KUKA KRL program: traccionv1.src, traccionv1.dat

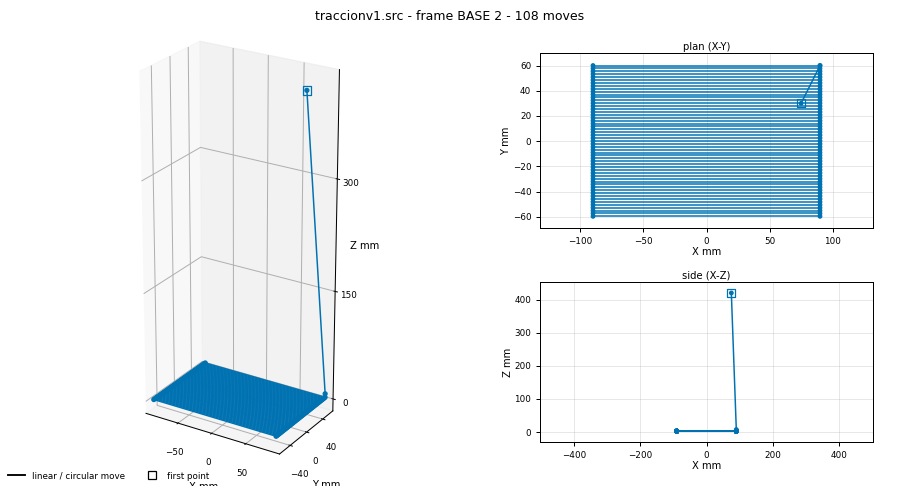
[picture p0: tool path of traccionv1.src in frame BASE 2, 108 of 110 moves have a stored position in this frame; points joined in program order, loops and branches not executed]
--- traccionv1.src ---
&ACCESS RVP
&PARAM TEMPLATE = C:\KRC\Roboter\Template\vorgabe
&PARAM EDITMASK = *
DEF traccionv1( )
;FOLD INI;%{PE}%V3.2.0,%MKUKATPBASIS,%CINIT,%VCOMMON,%P
;FOLD BAS INI;%{E}%V3.2.0,%MKUKATPBASIS,%CINIT,%VINIT,%P
GLOBAL INTERRUPT DECL 3 WHEN $STOPMESS==TRUE DO IR_STOPM ( )
INTERRUPT ON 3
BAS (#INITMOV,0 )
;ENDFOLD (BAS INI)
;FOLD A20 INI;%{E}%V3.2.0,%MKUKATPA20,%CINIT,%VINIT,%P
IF ARC20==TRUE THEN
A20 (ARC_INI)
INTERRUPT DECL 6 WHEN $CYCFLAG[3]==FALSE DO A20(TECH_STOP2)
ENDIF
;ENDFOLD (A20 INI)
;FOLD A10 INI;%{E}%V3.2.0,%MKUKATPARC,%CINIT,%VINIT,%P
IF A10_OPTION==#ACTIVE THEN
INTERRUPT DECL 4 WHEN $CYCFLAG[2]==FALSE DO A10 (#APPL_ERROR)
INTERRUPT DECL 7 WHEN A_ARC_SWI==#ACTIVE DO A10 (#ARC_SEAM)
INTERRUPT DECL 5 WHEN A_FLY_ARC==TRUE DO A10 (#HPU_ARC)
INTERRUPT  ON 5
A10_INI ( )
ENDIF
;ENDFOLD (A10 INI)
;FOLD GRIPPER INI;%{E}%V3.2.0,%MKUKATPGRIPPER,%CINIT,%VINIT,%P
USER_GRP(0,DUMMY,DUMMY,GDEFAULT)
;ENDFOLD (GRIPPER INI)
;FOLD SPOT INI;%{E}%V3.2.0,%MKUKATPSPOT,%CINIT,%VINIT,%P
USERSPOT(#INIT)
;ENDFOLD (SPOT INI)
;FOLD TOUCHSENSE INI;%{E}%V3.2.0,%MKUKATPTS,%CINIT,%VINIT,%P
IF H70_OPTION THEN
INTERRUPT DECL 15 WHEN $MEAS_PULSE[TOUCH_I[TOUCH_ACTIVE].IN_NR] DO H70 (6,CD0 )
INTERRUPT DECL 16 WHEN $ZERO_MOVE DO H70 (7,CD0 )
INTERRUPT DECL 17 WHEN $TECHPAR_C[FG_TOUCH,8]>0.5 DO H70 (8,CD0)
H70 (1,CD0 )
ENDIF
;ENDFOLD (TOUCHSENSE INI)
;FOLD USER INI;%{E}%V3.2.0,%MKUKATPUSER,%CINIT,%VINIT,%P
;Make your modifications here
;ENDFOLD (USER INI)
;ENDFOLD (INI)
; SPEED PTP FOR AXIS
$VEL_AXIS[1] = 15
$VEL_AXIS[2] = 15
$VEL_AXIS[3] = 15
$VEL_AXIS[4] = 15
$VEL_AXIS[5] = 15
$VEL_AXIS[6] = 15
;SMOOTHNESS
$APO.CDIS = 2
;ADVANCE
$ADVANCE = 3
;SET TOOL AND BASE
$TOOL = TOOL_DATA[3]
$BASE = BASE_DATA[2]
;HOME
;FOLD PTP HOME Vel=10% DEFAULT
$BWDSTART=FALSE
$H_POS=XHOME
PDAT_ACT=PDEFAULT
FDAT_ACT=FHOME
BAS(#PTP_DAT )
BAS (#VEL_PTP,10 )
PTP XHOME
;ENDFOLD
;USER PROGRAM
;SPEED $VEL.CP
$VEL.CP=0.045
; OUT[TEMP] = 200
; OUT[vent] = 1
; OUT[RPM] = 45
; USER POSES CALLS
PTP {X 75, Y 30, Z 420, A 0, B 90, C 0}
; USER POSES CALLS
LIN {X 90.0, Y 60.0, Z 7.5, A 0, B 90, C 0} C_DIS
WAIT SEC 1
$OUT[1] = TRUE
LIN {X 90.0, Y 60.0, Z 2.5, A 0, B 90, C 0} C_DIS
LIN {X -90.0, Y 60.0, Z 2.5, A 0, B 90, C 0} C_DIS
LIN {X -90.0, Y 57.7, Z 2.5, A 0, B 90, C 0} C_DIS
LIN {X 90.0, Y 57.7, Z 2.5, A 0, B 90, C 0} C_DIS
LIN {X 90.0, Y 55.4, Z 2.5, A 0, B 90, C 0} C_DIS
LIN {X -90.0, Y 55.4, Z 2.5, A 0, B 90, C 0} C_DIS
LIN {X -90.0, Y 53.1, Z 2.5, A 0, B 90, C 0} C_DIS
LIN {X 90.0, Y 53.1, Z 2.5, A 0, B 90, C 0} C_DIS
LIN {X 90.0, Y 50.8, Z 2.5, A 0, B 90, C 0} C_DIS
LIN {X -90.0, Y 50.8, Z 2.5, A 0, B 90, C 0} C_DIS
LIN {X -90.0, Y 48.5, Z 2.5, A 0, B 90, C 0} C_DIS
LIN {X 90.0, Y 48.5, Z 2.5, A 0, B 90, C 0} C_DIS
LIN {X 90.0, Y 46.2, Z 2.5, A 0, B 90, C 0} C_DIS
LIN {X -90.0, Y 46.2, Z 2.5, A 0, B 90, C 0} C_DIS
LIN {X -90.0, Y 43.9, Z 2.5, A 0, B 90, C 0} C_DIS
LIN {X 90.0, Y 43.9, Z 2.5, A 0, B 90, C 0} C_DIS
LIN {X 90.0, Y 41.6, Z 2.5, A 0, B 90, C 0} C_DIS
LIN {X -90.0, Y 41.6, Z 2.5, A 0, B 90, C 0} C_DIS
LIN {X -90.0, Y 39.3, Z 2.5, A 0, B 90, C 0} C_DIS
LIN {X 90.0, Y 39.3, Z 2.5, A 0, B 90, C 0} C_DIS
LIN {X 90.0, Y 37.0, Z 2.5, A 0, B 90, C 0} C_DIS
LIN {X -90.0, Y 37.0, Z 2.5, A 0, B 90, C 0} C_DIS
LIN {X -90.0, Y 34.7, Z 2.5, A 0, B 90, C 0} C_DIS
LIN {X 90.0, Y 34.7, Z 2.5, A 0, B 90, C 0} C_DIS
LIN {X 90.0, Y 32.4, Z 2.5, A 0, B 90, C 0} C_DIS
LIN {X -90.0, Y 32.4, Z 2.5, A 0, B 90, C 0} C_DIS
LIN {X -90.0, Y 30.1, Z 2.5, A 0, B 90, C 0} C_DIS
LIN {X 90.0, Y 30.1, Z 2.5, A 0, B 90, C 0} C_DIS
LIN {X 90.0, Y 27.8, Z 2.5, A 0, B 90, C 0} C_DIS
LIN {X -90.0, Y 27.8, Z 2.5, A 0, B 90, C 0} C_DIS
LIN {X -90.0, Y 25.5, Z 2.5, A 0, B 90, C 0} C_DIS
LIN {X 90.0, Y 25.5, Z 2.5, A 0, B 90, C 0} C_DIS
LIN {X 90.0, Y 23.2, Z 2.5, A 0, B 90, C 0} C_DIS
LIN {X -90.0, Y 23.2, Z 2.5, A 0, B 90, C 0} C_DIS
LIN {X -90.0, Y 20.9, Z 2.5, A 0, B 90, C 0} C_DIS
LIN {X 90.0, Y 20.9, Z 2.5, A 0, B 90, C 0} C_DIS
LIN {X 90.0, Y 18.6, Z 2.5, A 0, B 90, C 0} C_DIS
LIN {X -90.0, Y 18.6, Z 2.5, A 0, B 90, C 0} C_DIS
LIN {X -90.0, Y 16.3, Z 2.5, A 0, B 90, C 0} C_DIS
LIN {X 90.0, Y 16.3, Z 2.5, A 0, B 90, C 0} C_DIS
LIN {X 90.0, Y 14.0, Z 2.5, A 0, B 90, C 0} C_DIS
LIN {X -90.0, Y 14.0, Z 2.5, A 0, B 90, C 0} C_DIS
LIN {X -90.0, Y 11.7, Z 2.5, A 0, B 90, C 0} C_DIS
LIN {X 90.0, Y 11.7, Z 2.5, A 0, B 90, C 0} C_DIS
LIN {X 90.0, Y 9.4, Z 2.5, A 0, B 90, C 0} C_DIS
LIN {X -90.0, Y 9.4, Z 2.5, A 0, B 90, C 0} C_DIS
LIN {X -90.0, Y 7.1, Z 2.5, A 0, B 90, C 0} C_DIS
LIN {X 90.0, Y 7.1, Z 2.5, A 0, B 90, C 0} C_DIS
LIN {X 90.0, Y 4.8, Z 2.5, A 0, B 90, C 0} C_DIS
LIN {X -90.0, Y 4.8, Z 2.5, A 0, B 90, C 0} C_DIS
LIN {X -90.0, Y 2.5, Z 2.5, A 0, B 90, C 0} C_DIS
LIN {X 90.0, Y 2.5, Z 2.5, A 0, B 90, C 0} C_DIS
LIN {X 90.0, Y 0.2, Z 2.5, A 0, B 90, C 0} C_DIS
LIN {X -90.0, Y 0.2, Z 2.5, A 0, B 90, C 0} C_DIS
LIN {X -90.0, Y -2.1, Z 2.5, A 0, B 90, C 0} C_DIS
LIN {X 90.0, Y -2.1, Z 2.5, A 0, B 90, C 0} C_DIS
LIN {X 90.0, Y -4.4, Z 2.5, A 0, B 90, C 0} C_DIS
LIN {X -90.0, Y -4.4, Z 2.5, A 0, B 90, C 0} C_DIS
LIN {X -90.0, Y -6.7, Z 2.5, A 0, B 90, C 0} C_DIS
LIN {X 90.0, Y -6.7, Z 2.5, A 0, B 90, C 0} C_DIS
LIN {X 90.0, Y -9.0, Z 2.5, A 0, B 90, C 0} C_DIS
LIN {X -90.0, Y -9.0, Z 2.5, A 0, B 90, C 0} C_DIS
LIN {X -90.0, Y -11.3, Z 2.5, A 0, B 90, C 0} C_DIS
LIN {X 90.0, Y -11.3, Z 2.5, A 0, B 90, C 0} C_DIS
LIN {X 90.0, Y -13.6, Z 2.5, A 0, B 90, C 0} C_DIS
LIN {X -90.0, Y -13.6, Z 2.5, A 0, B 90, C 0} C_DIS
LIN {X -90.0, Y -15.9, Z 2.5, A 0, B 90, C 0} C_DIS
LIN {X 90.0, Y -15.9, Z 2.5, A 0, B 90, C 0} C_DIS
LIN {X 90.0, Y -18.2, Z 2.5, A 0, B 90, C 0} C_DIS
LIN {X -90.0, Y -18.2, Z 2.5, A 0, B 90, C 0} C_DIS
LIN {X -90.0, Y -20.5, Z 2.5, A 0, B 90, C 0} C_DIS
LIN {X 90.0, Y -20.5, Z 2.5, A 0, B 90, C 0} C_DIS
LIN {X 90.0, Y -22.8, Z 2.5, A 0, B 90, C 0} C_DIS
LIN {X -90.0, Y -22.8, Z 2.5, A 0, B 90, C 0} C_DIS
LIN {X -90.0, Y -25.1, Z 2.5, A 0, B 90, C 0} C_DIS
LIN {X 90.0, Y -25.1, Z 2.5, A 0, B 90, C 0} C_DIS
LIN {X 90.0, Y -27.4, Z 2.5, A 0, B 90, C 0} C_DIS
LIN {X -90.0, Y -27.4, Z 2.5, A 0, B 90, C 0} C_DIS
LIN {X -90.0, Y -29.7, Z 2.5, A 0, B 90, C 0} C_DIS
LIN {X 90.0, Y -29.7, Z 2.5, A 0, B 90, C 0} C_DIS
LIN {X 90.0, Y -32.0, Z 2.5, A 0, B 90, C 0} C_DIS
LIN {X -90.0, Y -32.0, Z 2.5, A 0, B 90, C 0} C_DIS
LIN {X -90.0, Y -34.3, Z 2.5, A 0, B 90, C 0} C_DIS
LIN {X 90.0, Y -34.3, Z 2.5, A 0, B 90, C 0} C_DIS
LIN {X 90.0, Y -36.6, Z 2.5, A 0, B 90, C 0} C_DIS
LIN {X -90.0, Y -36.6, Z 2.5, A 0, B 90, C 0} C_DIS
LIN {X -90.0, Y -38.9, Z 2.5, A 0, B 90, C 0} C_DIS
LIN {X 90.0, Y -38.9, Z 2.5, A 0, B 90, C 0} C_DIS
LIN {X 90.0, Y -41.2, Z 2.5, A 0, B 90, C 0} C_DIS
LIN {X -90.0, Y -41.2, Z 2.5, A 0, B 90, C 0} C_DIS
LIN {X -90.0, Y -43.5, Z 2.5, A 0, B 90, C 0} C_DIS
LIN {X 90.0, Y -43.5, Z 2.5, A 0, B 90, C 0} C_DIS
LIN {X 90.0, Y -45.8, Z 2.5, A 0, B 90, C 0} C_DIS
LIN {X -90.0, Y -45.8, Z 2.5, A 0, B 90, C 0} C_DIS
LIN {X -90.0, Y -48.1, Z 2.5, A 0, B 90, C 0} C_DIS
LIN {X 90.0, Y -48.1, Z 2.5, A 0, B 90, C 0} C_DIS
LIN {X 90.0, Y -50.4, Z 2.5, A 0, B 90, C 0} C_DIS
LIN {X -90.0, Y -50.4, Z 2.5, A 0, B 90, C 0} C_DIS
LIN {X -90.0, Y -52.7, Z 2.5, A 0, B 90, C 0} C_DIS
LIN {X 90.0, Y -52.7, Z 2.5, A 0, B 90, C 0} C_DIS
LIN {X 90.0, Y -55.0, Z 2.5, A 0, B 90, C 0} C_DIS
LIN {X -90.0, Y -55.0, Z 2.5, A 0, B 90, C 0} C_DIS
LIN {X -90.0, Y -57.3, Z 2.5, A 0, B 90, C 0} C_DIS
LIN {X 90.0, Y -57.3, Z 2.5, A 0, B 90, C 0} C_DIS
LIN {X 90.0, Y -59.6, Z 2.5, A 0, B 90, C 0} C_DIS
LIN {X -90.0, Y -59.6, Z 2.5, A 0, B 90, C 0} C_DIS
$OUT[1] = FALSE

;Wait for
; END POSITION FOR
;END USER CODE
;HOME
;FOLD PTP HOME Vel=10% DEFAULT
$BWDSTART=FALSE
$H_POS=XHOME
PDAT_ACT=PDEFAULT
FDAT_ACT=FHOME
BAS(#PTP_DAT )
BAS (#VEL_PTP,10 )
PTP XHOME
;ENDFOLD
END

--- traccionv1.dat ---
DEFDAT traccionv1()
ENDDAT
